// TIA Portal V20 export
FUNCTION "PostProcessing" : Void   // FC57, LAD
TITLE = Post Processing
// V1.0  25.05.04  Safety test program: sending data via F-link
// stored: Namespace Safety, SetENOAutomatically false
BEGIN

REGION Network 1: Sending data to BA010, ReelCut #1
   // V1.0  25.05.04  Safety test program: FlinkSendToBA10AC1
   //                 Send ID: 130, Receive ID: 131
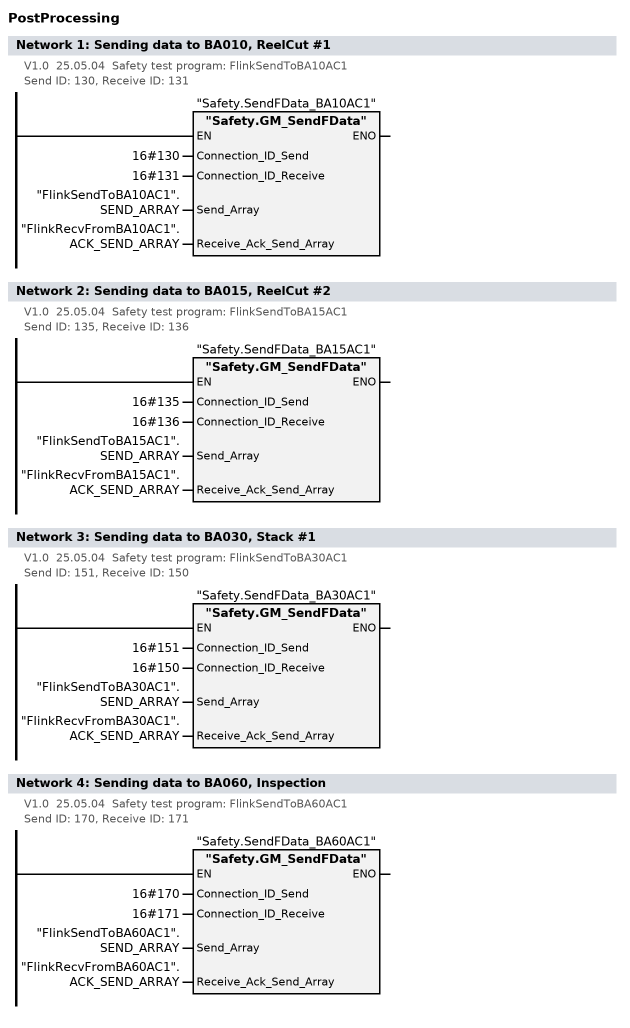
   RUNG wire#powerrail
      "Safety.SendFData_BA10AC1"(Connection_ID_Send := 16#130, Connection_ID_Receive := 16#131, Send_Array := "FlinkSendToBA10AC1".SEND_ARRAY, Receive_Ack_Send_Array := "FlinkRecvFromBA10AC1".ACK_SEND_ARRAY)
   END_RUNG
   // the same network as SCL:
   "Safety.SendFData_BA10AC1"(Connection_ID_Send := 16#130,   // "Safety.GM_SendFData"
                           Connection_ID_Receive := 16#131,
                           Send_Array := "FlinkSendToBA10AC1".SEND_ARRAY,
                           Receive_Ack_Send_Array := "FlinkRecvFromBA10AC1".ACK_SEND_ARRAY);
END_REGION

REGION Network 2: Sending data to BA015, ReelCut #2
   // V1.0  25.05.04  Safety test program: FlinkSendToBA15AC1
   //                 Send ID: 135, Receive ID: 136
   RUNG wire#powerrail
      "Safety.SendFData_BA15AC1"(Connection_ID_Send := 16#135, Connection_ID_Receive := 16#136, Send_Array := "FlinkSendToBA15AC1".SEND_ARRAY, Receive_Ack_Send_Array := "FlinkRecvFromBA15AC1".ACK_SEND_ARRAY)
   END_RUNG
   // the same network as SCL:
   "Safety.SendFData_BA15AC1"(Connection_ID_Send := 16#135,   // "Safety.GM_SendFData"
                           Connection_ID_Receive := 16#136,
                           Send_Array := "FlinkSendToBA15AC1".SEND_ARRAY,
                           Receive_Ack_Send_Array := "FlinkRecvFromBA15AC1".ACK_SEND_ARRAY);
END_REGION

REGION Network 3: Sending data to BA030, Stack #1
   // V1.0  25.05.04  Safety test program: FlinkSendToBA30AC1
   //                 Send ID: 151, Receive ID: 150
   RUNG wire#powerrail
      "Safety.SendFData_BA30AC1"(Connection_ID_Send := 16#151, Connection_ID_Receive := 16#150, Send_Array := "FlinkSendToBA30AC1".SEND_ARRAY, Receive_Ack_Send_Array := "FlinkRecvFromBA30AC1".ACK_SEND_ARRAY)
   END_RUNG
   // the same network as SCL:
   "Safety.SendFData_BA30AC1"(Connection_ID_Send := 16#151,   // "Safety.GM_SendFData"
                           Connection_ID_Receive := 16#150,
                           Send_Array := "FlinkSendToBA30AC1".SEND_ARRAY,
                           Receive_Ack_Send_Array := "FlinkRecvFromBA30AC1".ACK_SEND_ARRAY);
END_REGION

REGION Network 4: Sending data to BA060, Inspection
   // V1.0  25.05.04  Safety test program: FlinkSendToBA60AC1
   //                 Send ID: 170, Receive ID: 171
   RUNG wire#powerrail
      "Safety.SendFData_BA60AC1"(Connection_ID_Send := 16#170, Connection_ID_Receive := 16#171, Send_Array := "FlinkSendToBA60AC1".SEND_ARRAY, Receive_Ack_Send_Array := "FlinkRecvFromBA60AC1".ACK_SEND_ARRAY)
   END_RUNG
   // the same network as SCL:
   "Safety.SendFData_BA60AC1"(Connection_ID_Send := 16#170,   // "Safety.GM_SendFData"
                           Connection_ID_Receive := 16#171,
                           Send_Array := "FlinkSendToBA60AC1".SEND_ARRAY,
                           Receive_Ack_Send_Array := "FlinkRecvFromBA60AC1".ACK_SEND_ARRAY);
END_REGION

REGION Network 5 (SCL): Set ACK_OP value in DataToSafety
   //Set ACK_OP value in DataToSafety DB
   "Safety.DataToSafety".ackSafetyFromHmi := "Safety.DataFromStandard".ackSafetyFromHmi;
   "Safety.DataFromSafety".ackOP_changeRequired := "Safety.InstMain_Safety_RTG1".instAckOP.Q;
END_REGION
END_FUNCTION
